FUNCTION_BLOCK T_AxisComponent EXTENDS FB_ComponentBase IMPLEMENTS I_AxisComponent
VAR
	_axis: I_Axis;
END_VAR

METHOD GenericInitialise
VAR_INPUT
	Axis : I_Axis;
END_VAR
_axis := Axis;
END_METHOD

END_FUNCTION_BLOCK

(* stored: Version 1.1.0.1, ProductVersion 3.1.4024.12
   POU T_AxisComponent: Id {0fe96c03-9172-44c6-9878-730cd9cf8c50}, SpecialFunc None
   Method GenericInitialise: Id {4c8e05c1-d10b-4975-ac2b-01709bb89536} *)
